FUNCTION_BLOCK MOD_OccupationLogic (* Occupation by session ID: Occupy when free (or again by the owner), Release only by the owner *)
  (* Standard: 61499-2 *)
  (* Version 0.1, 2026-09-28, Project contributors, AAU Smart Production Lab *)
  PACKAGE modlib;
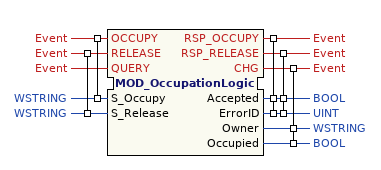
  EVENT_INPUT
    OCCUPY WITH S_Occupy;
    RELEASE WITH S_Release;
    QUERY;
  END_EVENT
  EVENT_OUTPUT
    RSP_OCCUPY WITH Accepted, ErrorID;
    RSP_RELEASE WITH Accepted, ErrorID;
    CHG WITH Owner, Occupied;
  END_EVENT
  VAR_INPUT
    S_Occupy : WSTRING;
    S_Release : WSTRING;
  END_VAR
  VAR_OUTPUT
    Accepted : BOOL;
    ErrorID : UINT;
    Owner : WSTRING;
    Occupied : BOOL;
  END_VAR
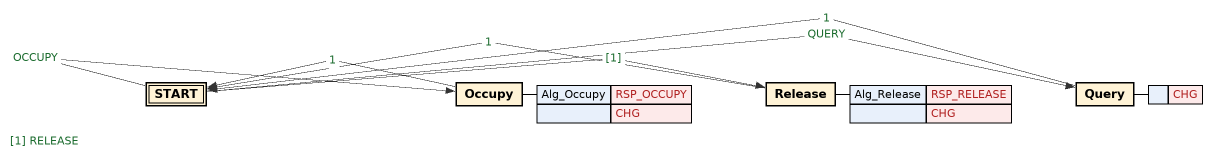
  EC_STATES
    START;
    Occupy : Alg_Occupy -> RSP_OCCUPY, -> CHG;
    Release : Alg_Release -> RSP_RELEASE, -> CHG;
    Query : -> CHG;
  END_STATES
  EC_TRANSITIONS
    START TO Occupy := OCCUPY;
    Occupy TO START := 1;
    START TO Release := RELEASE;
    Release TO START := 1;
    START TO Query := QUERY;
    Query TO START := 1;
  END_TRANSITIONS
  ALGORITHM Alg_Occupy IN ST:
IF (S_Occupy <> "") AND ((Owner = "") OR (Owner = S_Occupy)) THEN
  Owner := S_Occupy;
  Occupied := TRUE;
  Accepted := TRUE;
  ErrorID := 0;
ELSE
  Accepted := FALSE;
  ErrorID := 5;
END_IF;
  END_ALGORITHM
  ALGORITHM Alg_Release IN ST:
IF (Owner <> "") AND (Owner = S_Release) THEN
  Owner := "";
  Occupied := FALSE;
  Accepted := TRUE;
  ErrorID := 0;
ELSE
  Accepted := FALSE;
  ErrorID := 5;
END_IF;
  END_ALGORITHM
END_FUNCTION_BLOCK
